{attribute 'linkalways'} 
{attribute 'no_explicit_call' := 'This FB is a CLASS and must be accessed using methods or properties'}
{attribute 'enable_dynamic_creation'}
FUNCTION_BLOCK Queue EXTENDS Disposable IMPLEMENTS I_Queue
VAR
	linkedList : LinkedList;
END_VAR

METHOD AddItem
VAR_INPUT
	Item : ANY;
END_VAR
Enqueue(Item);
END_METHOD

METHOD PUBLIC Clear
VAR_INPUT
END_VAR
linkedList.Clear();
END_METHOD

METHOD PUBLIC Contains : BOOL;
VAR_INPUT
	Item : ANY;
END_VAR
VAR
	found : I_LinkedListNode;
END_VAR
found := linkedList.Find(Item);
Contains := found <> 0;
END_METHOD

METHOD PUBLIC CopyTo : BOOL
VAR_INPUT
	Destination : ANY;
END_VAR
CopyTo := linkedList.CopyTo(Destination);
END_METHOD

METHOD PUBLIC CopyToLocation : BOOL
VAR_INPUT
	Destination : PVOID;
	DestinationSize : UDINT;
END_VAR
CopyToLocation := linkedList.CopyToLocation(Destination,DestinationSize);
END_METHOD

PROPERTY PUBLIC Count : ULINT
GET
Count := linkedList.Count;
END_GET
END_PROPERTY

METHOD PUBLIC Enqueue
VAR_INPUT
	Item : ANY;
END_VAR
linkedList.AddLast(Item);
END_METHOD

METHOD FB_exit : BOOL
VAR_INPUT
	bInCopyCode : BOOL; // if TRUE, the exit method is called for exiting an instance that is copied afterwards (online change).
END_VAR
IF bInCopyCode THEN
	RETURN;
END_IF

Clear();
END_METHOD

METHOD PUBLIC GetEnumerator : I_ForwardEnumerator
GetEnumerator := linkedList.GetEnumerator();
END_METHOD

METHOD RemoveItem : BOOL
VAR_INPUT
	Item : ANY;
END_VAR
RemoveItem := linkedList.RemoveItem(Item);
END_METHOD

METHOD PUBLIC TryDequeue : BOOL;
VAR_INPUT
	Destination : ANY;
END_VAR
VAR
	first : I_LinkedListNode;
	dequeued : BOOL;
END_VAR
first := linkedList.First;

IF first = 0 THEN
	RETURN;
END_IF

dequeued := linkedList.First.Get(Destination);

IF NOT dequeued THEN
	RETURN;
END_IF

linkedList.RemoveFirst();
TryDequeue := TRUE;
END_METHOD

METHOD PUBLIC TryPeek : BOOL;
VAR_INPUT
	Destination : ANY;
END_VAR
VAR
	first : I_LinkedListNode;
END_VAR
first := linkedList.First;

IF first = 0 THEN
	RETURN;
END_IF

TryPeek := first.Get(Destination);
END_METHOD

END_FUNCTION_BLOCK

(* stored: Version 1.1.0.1, ProductVersion 3.1.4024.12
   POU Queue: Id {60047339-337c-4be5-ae72-2dad2c213009}, SpecialFunc None
   Folder Destructor: Id {62d87962-2cf7-4a17-898b-21ae6a43eedf}
   Method AddItem: Id {50300d84-c466-44f9-ac93-88f7eb39d43d}
   Method Clear: Id {be525374-c8c0-4800-8d21-3dedb89b7102}
   Method Contains: Id {41c5234e-0ba0-4792-9541-46f8eba2e5bf}
   Method CopyTo: Id {da75c79e-2f53-47df-bd3d-75645cba429f}
   Method CopyToLocation: Id {c0c023f3-1e5b-4896-b6fb-35b8f504ba53}
   Property Count: Id {a5b5dc0d-9136-4d33-8a44-3fd5f4753277}
   Get Get: Id {3a2945f3-109a-481b-88d2-6b143645dca6}
   Method Enqueue: Id {55f220d0-7765-476a-8e45-859c45790653}
   Method FB_exit: Id {7b2a3bda-d078-45e7-a397-f44960e647ab}
   Method GetEnumerator: Id {313bc49e-d42c-4e4f-9245-f744dca425c4}
   Method RemoveItem: Id {8d5fb1bb-9563-472f-98a8-85ffcecd9667}
   Method TryDequeue: Id {6a1352f2-9546-44f6-a541-e9c3fd20ae65}
   Method TryPeek: Id {c32c66c4-721d-4fa4-8a6a-dc6c4b397149} *)
